FUNCTION_BLOCK FB_MessageLinkedList EXTENDS FB_GenericLinkedList
VAR_INPUT
END_VAR
VAR_OUTPUT
END_VAR
VAR
END_VAR

METHOD M_AddMessageToHead : BOOL
VAR_INPUT
	pUnitToAdd : POINTER TO ST_LinkedListUnit;
	pMessageToAdd : POINTER TO ST_Message;
END_VAR
pUnitToAdd^.pVoid := pMessageToAdd;
SUPER^.M_AddToHead(pUnitToAdd);
END_METHOD

METHOD M_AddMessageToTail : BOOL
VAR_INPUT
	pUnitToAdd : POINTER TO ST_LinkedListUnit;
	pMessageToAdd : POINTER TO ST_Message;
END_VAR
pUnitToAdd^.pVoid := pMessageToAdd;
SUPER^.M_AddToTail(pUnitToAdd);
END_METHOD

METHOD M_GetHeadMessage : POINTER TO ST_Message
VAR_INPUT
END_VAR
VAR
	stUnit : POINTER TO ST_LinkedListUnit;
END_VAR
stUnit := SUPER^.M_GetHead();

IF stUnit = NULL THEN
	RETURN;
END_IF

M_GetHeadMessage := stUnit^.pVoid;
END_METHOD

METHOD M_GetNextMessage : POINTER TO ST_Message
VAR
	stUnit : POINTER TO ST_LinkedListUnit;
END_VAR
stUnit := SUPER^.M_GetNext();

IF stUnit = NULL THEN
	RETURN;
END_IF

M_GetNextMessage := stUnit^.pVoid;
END_METHOD

METHOD M_GetTailMessage : POINTER TO ST_Message
VAR_INPUT
END_VAR
VAR
	stUnit : POINTER TO ST_LinkedListUnit;

END_VAR
stUnit := SUPER^.M_GetTail();

IF stUnit = NULL THEN
	RETURN;
END_IF

M_GetTailMessage := stUnit^.pVoid;
END_METHOD

END_FUNCTION_BLOCK

(* stored: Version 1.1.0.1, ProductVersion 3.1.4022.16
   POU FB_MessageLinkedList: Id {0a675e83-a9f7-478c-a06d-302d55c7e31e}, SpecialFunc None
   Method M_AddMessageToHead: Id {ae86983b-ba05-4b50-b320-34d1277b4b1c}
   Method M_AddMessageToTail: Id {1d371728-ade8-492b-b36e-6c54ca1c2f22}
   Method M_GetHeadMessage: Id {8e0c366b-4593-453a-b33d-c3a611a6d960}
   Method M_GetNextMessage: Id {6aa4a480-4c10-4662-a778-e37cf54a11ac}
   Method M_GetTailMessage: Id {fb54e427-3cac-40e4-9bca-d1112e937033} *)
